TYPE ST_Error :
STRUCT
	nErrorID  	: INT;
	ErrorTime 	: DT;
	ErrorStatus : BOOL;
END_STRUCT
END_TYPE

(* stored: Version 1.1.0.1, ProductVersion 3.1.4024.12
   DUT ST_Error: Id {d47ce2c4-8dcb-4624-9241-ee58dfb00dc9} *)
